// TIA Portal V21 export
VAR_GLOBAL   // PLC tag table "Pid_PhysicalQuantity"
END_VAR
VAR_GLOBAL CONSTANT   // user constants
   Pid_PhysicalQuantity_Percentuale : Int := 0;
   Pid_PhysicalQuantity_Pressione : Int := 2;
   Pid_PhysicalQuantity_Lunghezza : Int := 3;
   Pid_PhysicalQuantity_Portata : Int := 4;
   Pid_PhysicalQuantity_Luminosità : Int := 5;
   Pid_PhysicalQuantity_GradoIlluminazione : Int := 6;
   Pid_PhysicalQuantity_Forza : Int := 7;
   Pid_PhysicalQuantity_CoppiaSerraggio : Int := 8;
   Pid_PhysicalQuantity_Massa : Int := 9;
   Pid_PhysicalQuantity_Corrente : Int := 10;
   Pid_PhysicalQuantity_Tensione : Int := 11;
   Pid_PhysicalQuantity_Potenza : Int := 12;
   Pid_PhysicalQuantity_Superficie : Int := 13;
   Pid_PhysicalQuantity_Temperatura : Int := 1;
   Pid_PhysicalQuantity_Volume : Int := 14;
   Pid_PhysicalQuantity_Angolo : Int := 15;
   Pid_PhysicalQuantity_Viscosità : Int := 16;
   Pid_PhysicalQuantity_NumeroGiri : Int := 17;
   Pid_PhysicalQuantity_Velocità : Int := 18;
   Pid_PhysicalQuantity_Spessore : Int := 19;
   Pid_PhysicalQuantity_Frequenza : Int := 20;
   Pid_PhysicalQuantity_VelocitàAngolare : Int := 21;
END_VAR
